{attribute 'qualified_only'}
{attribute 'strict'}
{attribute 'to_string'}
TYPE E_Barcode_State :
(
	INIT := 0,
	SEND_POS_VEL_COMMAND := 10,
	SEND_DIAGNOSTIC_COMMAND := 20,
	SEND_MARKER_INFO_COMMAND := 30,
	ERROR := 999
);
END_TYPE

(* stored: Version 1.1.0.1
   DUT E_Barcode_State: Id {fe91f11c-2bd7-4302-af1e-48ee1b668ab0} *)
